FUNCTION_BLOCK FB_AxisReadParams
VAR_INPUT
	bExecute: BOOL;
	bReset: BOOL;
	stHardware: ST_AxisHardware;
END_VAR
VAR_OUTPUT
	stConfig: ST_AxisParams;
	bValid: BOOL;
	bBusy: BOOL;
	bError: BOOL;
	nErrorID: UDINT;
END_VAR
VAR_IN_OUT
	Axis: AXIS_REF;
END_VAR
VAR
	fbNCRead: FB_AxisReadNC;
	fbCoERead: FB_AxisReadCoE;
END_VAR

fbNCRead(bExecute:=bExecute,
	bReset:=bReset,
	stConfig:=stConfig,
	Axis:=Axis);
fbCoERead(bExecute:=bExecute,
	bReset:=bReset,
	stHardware:=stHardware,
	stConfig:=stConfig,
	Axis:=Axis);
bValid := fbNCRead.bValid AND NOT fbCoERead.bBusy AND NOT fbCoERead.bError AND bExecute;
bBusy := fbNCRead.bBusy OR fbCoERead.bBusy;
bError := fbNCRead.bError OR fbCoERead.bError;
IF fbNCRead.nErrorID > 0 THEN
	nErrorID := fbNCRead.nErrorID;
ELSE
	nErrorID := fbCoERead.nErrorID;
END_IF

END_FUNCTION_BLOCK

(* stored: Version 1.1.0.1, ProductVersion 3.1.4020.14
   POU FB_AxisReadParams: Id {e92502d6-67ee-4fa0-a7de-4596fc050760}, SpecialFunc None *)
